(* CODESYS project FU_sPaddFront.xml

Project tree, tasks and I/O mapping:
  function FU_sPaddFront [ST]
*)

// FU_sPaddFront
//This function padds the front of a string with the given character, the given amount
//If the padd amount plus the string is longer than the output string, the input string will be cut off to make space for the padding
// +-----------+----------+----------+-----------------------------------------------------------------------------------------------------------------------+
// |**Version**|**Author**| **Date** |**Changes**                                                                                                            |
// +-----------+----------+----------+-----------------------------------------------------------------------------------------------------------------------+
// | 1         | NSN      | 04-02-19 | Creation                                                                                                              |
// +-----------+----------+----------+-----------------------------------------------------------------------------------------------------------------------+
FUNCTION FU_sPaddFront : STRING(255)
VAR_INPUT
	sStr		:STRING(255);		//Input String
	wPadds		:WORD;				//How much to padd it
	eChar		:EASCII;		//Which character to padd with
END_VAR

FU_sPaddFrontBIBO(sOut:=FU_sPaddFront,sStr:=sStr,wPadds:=wPadds,wOutSize:=255,eChar:=eChar);

END_FUNCTION
